{attribute 'qualified_only'}
{attribute 'strict'}
TYPE E_MachineState :
(
	Critical,				//クリティカルの発生
	Error,					//エラーの発生
	Warning,				//ワーニングの発生
	Stay,					//McPowerがOFF
	Stop,					//McPowerがON
	Moving					//軸動作中
);
END_TYPE

(* stored: Version 1.1.0.1, ProductVersion 3.1.4026.12
   DUT E_MachineState: Id {b577c7d7-176f-4952-a6b4-4f333edaf8f8} *)
